FUNCTION_BLOCK SYSTEM_TIME (* Service Interface Function Block Type *)
  (* Standard: 61499-2 *)
  (* Version 0.0, 20/07/2021, josef, nxtControl GmBH, template *)
  PACKAGE Flexbridge.Iceblock;
  (* Compiler Cpp nxtControl builtin 1.0 *)
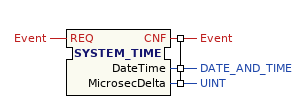
  EVENT_INPUT
    REQ; (* Service Request *)
  END_EVENT
  EVENT_OUTPUT
    CNF WITH DateTime, MicrosecDelta; (* Confirmation of Requested Service *)
  END_EVENT
  VAR_OUTPUT
    DateTime : DATE_AND_TIME;
    MicrosecDelta : UINT;
  END_VAR
  SERVICE SYSTEM_TIME/RESOURCE
    SEQUENCE normal_establishment
      SYSTEM_TIME.INIT+(PARAMS) -> RESOURCE.initialize(PARAMS) -> SYSTEM_TIME.INITO+();
    END_SEQUENCE
    SEQUENCE unsuccessful_establishment
      SYSTEM_TIME.INIT+(PARAMS) -> RESOURCE.initialize(PARAMS) -> SYSTEM_TIME.INITO-(STATUS);
    END_SEQUENCE
    SEQUENCE request_confirm
      SYSTEM_TIME.REQ+(SD) -> RESOURCE.request(SD) -> SYSTEM_TIME.CNF+(RD);
    END_SEQUENCE
    SEQUENCE request_inhibited
      SYSTEM_TIME.REQ-(SD) -> SYSTEM_TIME.CNF-(STATUS);
    END_SEQUENCE
    SEQUENCE request_error
      SYSTEM_TIME.REQ+(SD) -> RESOURCE.request(SD) -> SYSTEM_TIME.CNF-(STATUS);
    END_SEQUENCE
    SEQUENCE indication_response
      RESOURCE.indicate(RD) -> SYSTEM_TIME.IND+(RD);
      SYSTEM_TIME.RSP(QI,SD) -> RESOURCE.response(QI,SD);
    END_SEQUENCE
    SEQUENCE indication_inhibited
      RESOURCE.indicate(RD,QI=FALSE) -> RESOURCE.inhibited();
    END_SEQUENCE
    SEQUENCE error_indication
      RESOURCE.error(STATUS) -> SYSTEM_TIME.IND-(STATUS);
    END_SEQUENCE
    SEQUENCE application_initiated_termination
      SYSTEM_TIME.INIT-() -> RESOURCE.terminate() -> SYSTEM_TIME.INITO-(STATUS);
    END_SEQUENCE
    SEQUENCE resource_initiated_termination
      -> SYSTEM_TIME.INITO-(STATUS);
    END_SEQUENCE
  END_SERVICE
END_FUNCTION_BLOCK
